// TIA Portal V19 export
FUNCTION_BLOCK "Main Control"   // FB1, LAD
{ S7_Optimized_Access := 'TRUE' }
// stored: MemoryReserve 100, SetENOAutomatically false
   VAR
      store : Bool;
   END_VAR
   VAR_TEMP   // added for the SCL form of the ladder/FBD networks
      _w1 : Bool;
      _w2 : Bool;
   END_VAR
BEGIN

REGION Network 1: Control Auto Run
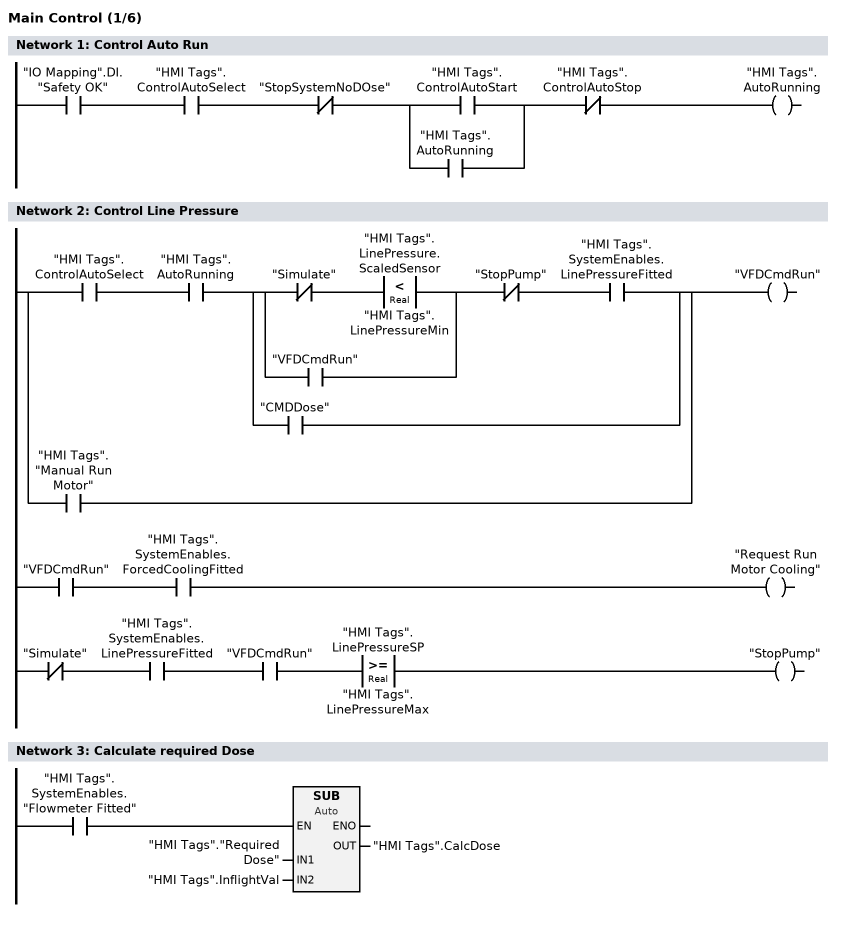
   RUNG wire#powerrail
      Contact( "IO Mapping".DI."Safety OK" )
      Contact( "HMI Tags".ControlAutoSelect )
      I_Contact( "StopSystemNoDOse" )
      wire#w1
      Contact( "HMI Tags".ControlAutoStart )
      wire#w2
      I_Contact( "HMI Tags".ControlAutoStop )
      Coil( "HMI Tags".AutoRunning )
   END_RUNG
   RUNG wire#w1
      Contact( "HMI Tags".AutoRunning )
   END_RUNG wire#w2
   // the same network as SCL:
   "HMI Tags".AutoRunning := "IO Mapping".DI."Safety OK" AND "HMI Tags".ControlAutoSelect AND NOT "StopSystemNoDOse" AND ("HMI Tags".ControlAutoStart OR "HMI Tags".AutoRunning) AND NOT "HMI Tags".ControlAutoStop;
END_REGION

REGION Network 2: Control Line Pressure
   RUNG wire#powerrail
      Contact( "HMI Tags".ControlAutoSelect )
      Contact( "HMI Tags".AutoRunning )
      wire#w1
      I_Contact( "Simulate" )
      { S7_Templates := "SrcType := Real" } LT_Contact(in1 := "HMI Tags".LinePressure.ScaledSensor, in2 := "HMI Tags".LinePressureMin)
      wire#w2
      I_Contact( "StopPump" )
      Contact( "HMI Tags".SystemEnables.LinePressureFitted )
      wire#w3
      Coil( "VFDCmdRun" )
   END_RUNG
   RUNG wire#w1
      Contact( "VFDCmdRun" )
   END_RUNG wire#w2
   RUNG wire#w1
      Contact( "CMDDose" )
   END_RUNG wire#w3
   RUNG wire#powerrail
      Contact( "HMI Tags"."Manual Run Motor" )
   END_RUNG wire#w3
   RUNG wire#powerrail
      Contact( "VFDCmdRun" )
      Contact( "HMI Tags".SystemEnables.ForcedCoolingFitted )
      Coil( "Request Run Motor Cooling" )
   END_RUNG
   RUNG wire#powerrail
      I_Contact( "Simulate" )
      Contact( "HMI Tags".SystemEnables.LinePressureFitted )
      Contact( "VFDCmdRun" )
      { S7_Templates := "SrcType := Real" } GE_Contact(in1 := "HMI Tags".LinePressureSP, in2 := "HMI Tags".LinePressureMax)
      Coil( "StopPump" )
   END_RUNG
   // the same network as SCL:
   "VFDCmdRun" := ("HMI Tags".ControlAutoSelect AND "HMI Tags".AutoRunning AND ((((NOT "Simulate" AND ("HMI Tags".LinePressure.ScaledSensor < "HMI Tags".LinePressureMin)) OR "VFDCmdRun") AND NOT "StopPump" AND "HMI Tags".SystemEnables.LinePressureFitted) OR "CMDDose")) OR "HMI Tags"."Manual Run Motor";
   "Request Run Motor Cooling" := "VFDCmdRun" AND "HMI Tags".SystemEnables.ForcedCoolingFitted;
   "StopPump" := NOT "Simulate" AND "HMI Tags".SystemEnables.LinePressureFitted AND "VFDCmdRun" AND ("HMI Tags".LinePressureSP >= "HMI Tags".LinePressureMax);
END_REGION

REGION Network 3: Calculate required Dose
   RUNG wire#powerrail
      Contact( "HMI Tags".SystemEnables."Flowmeter Fitted" )
      Sub(in1 := "HMI Tags"."Required Dose", in2 := "HMI Tags".InflightVal, out => "HMI Tags".CalcDose)
   END_RUNG
   // the same network as SCL:
   IF "HMI Tags".SystemEnables."Flowmeter Fitted" THEN
       "HMI Tags".CalcDose := "HMI Tags"."Required Dose" - "HMI Tags".InflightVal;
   END_IF;
END_REGION

REGION Network 4: Open Valves to Dose
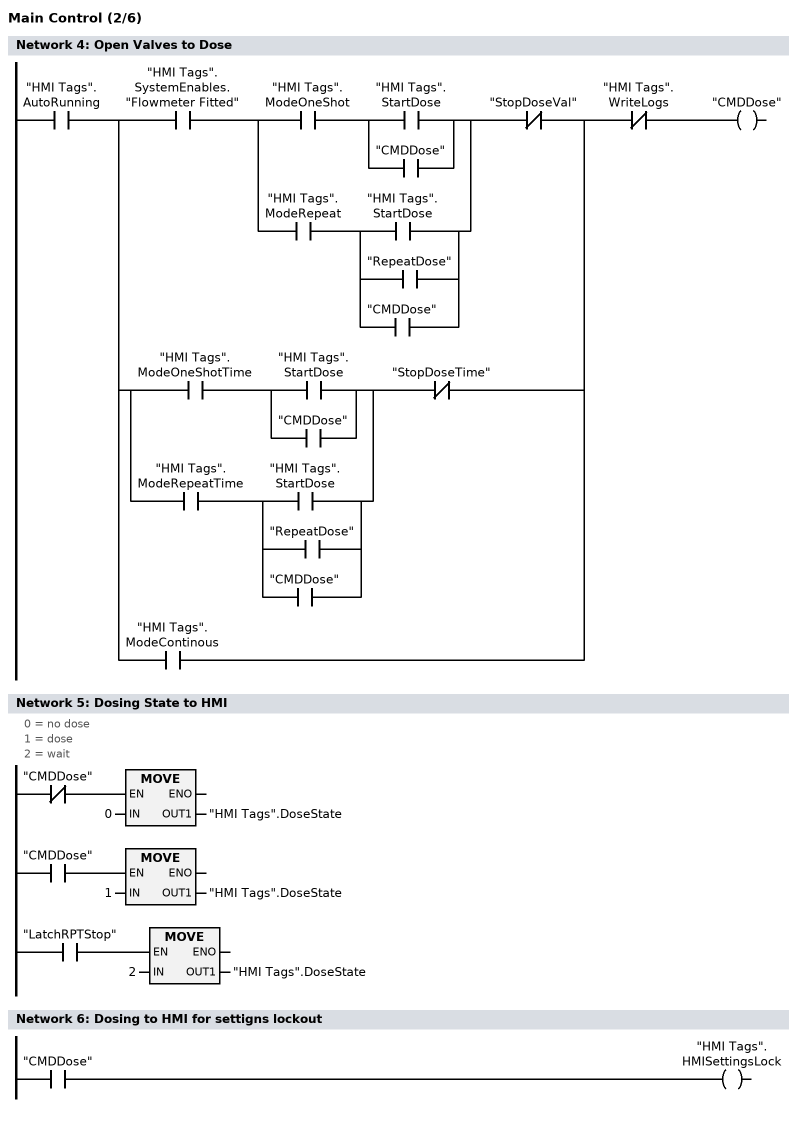
   RUNG wire#powerrail
      Contact( "HMI Tags".AutoRunning )
      wire#w1
      Contact( "HMI Tags".SystemEnables."Flowmeter Fitted" )
      wire#w2
      Contact( "HMI Tags".ModeOneShot )
      wire#w3
      Contact( "HMI Tags".StartDose )
      wire#w4
      I_Contact( "StopDoseVal" )
      wire#w6
      I_Contact( "HMI Tags".WriteLogs )
      Coil( "CMDDose" )
   END_RUNG
   RUNG wire#w3
      Contact( "CMDDose" )
   END_RUNG wire#w4
   RUNG wire#w2
      Contact( "HMI Tags".ModeRepeat )
      wire#w5
      Contact( "HMI Tags".StartDose )
   END_RUNG wire#w4
   RUNG wire#w5
      Contact( "RepeatDose" )
   END_RUNG wire#w4
   RUNG wire#w5
      Contact( "CMDDose" )
   END_RUNG wire#w4
   RUNG wire#w1
      Contact( "HMI Tags".ModeOneShotTime )
      wire#w7
      Contact( "HMI Tags".StartDose )
      wire#w8
      I_Contact( "StopDoseTime" )
   END_RUNG wire#w6
   RUNG wire#w7
      Contact( "CMDDose" )
   END_RUNG wire#w8
   RUNG wire#w1
      Contact( "HMI Tags".ModeRepeatTime )
      wire#w9
      Contact( "HMI Tags".StartDose )
   END_RUNG wire#w8
   RUNG wire#w9
      Contact( "RepeatDose" )
   END_RUNG wire#w8
   RUNG wire#w9
      Contact( "CMDDose" )
   END_RUNG wire#w8
   RUNG wire#w1
      Contact( "HMI Tags".ModeContinous )
   END_RUNG wire#w6
   // the same network as SCL:
   "CMDDose" := "HMI Tags".AutoRunning AND (("HMI Tags".SystemEnables."Flowmeter Fitted" AND (("HMI Tags".ModeOneShot AND ("HMI Tags".StartDose OR "CMDDose")) OR ("HMI Tags".ModeRepeat AND ("HMI Tags".StartDose OR "RepeatDose" OR "CMDDose"))) AND NOT "StopDoseVal") OR ((("HMI Tags".ModeOneShotTime AND ("HMI Tags".StartDose OR "CMDDose")) OR ("HMI Tags".ModeRepeatTime AND ("HMI Tags".StartDose OR "RepeatDose" OR "CMDDose"))) AND NOT "StopDoseTime") OR "HMI Tags".ModeContinous) AND NOT "HMI Tags".WriteLogs;
END_REGION

REGION Network 5: Dosing State to HMI
   // 0 = no dose
   // 1 = dose
   // 2 = wait
   RUNG wire#powerrail
      I_Contact( "CMDDose" )
      Move(in := 0, out1 => "HMI Tags".DoseState)
   END_RUNG
   RUNG wire#powerrail
      Contact( "CMDDose" )
      Move(in := 1, out1 => "HMI Tags".DoseState)
   END_RUNG
   RUNG wire#powerrail
      Contact( "LatchRPTStop" )
      Move(in := 2, out1 => "HMI Tags".DoseState)
   END_RUNG
   // the same network as SCL:
   IF NOT "CMDDose" THEN "HMI Tags".DoseState := 0; END_IF;
   IF "CMDDose" THEN "HMI Tags".DoseState := 1; END_IF;
   IF "LatchRPTStop" THEN "HMI Tags".DoseState := 2; END_IF;
END_REGION

REGION Network 6: Dosing to HMI for settigns lockout
   RUNG wire#powerrail
      Contact( "CMDDose" )
      Coil( "HMI Tags".HMISettingsLock )
   END_RUNG
   // the same network as SCL:
   "HMI Tags".HMISettingsLock := "CMDDose";
END_REGION

REGION Network 7: Command the flowmeter to count
   // This should start the flowmeter counting slightly ahead of opening the valves.
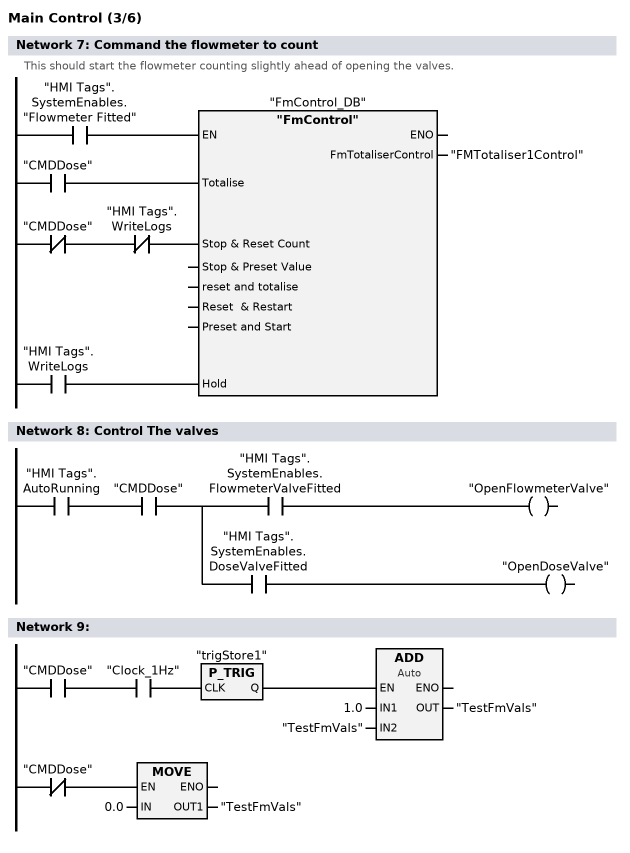
   RUNG wire#powerrail
      Contact( "HMI Tags".SystemEnables."Flowmeter Fitted" )
      "FmControl_DB"(Totalise := wire#w1, "Stop & Reset Count" := wire#w2, Hold := wire#w3, "Stop & Preset Value" :=, "reset and totalise" :=, "Reset  & Restart" :=, "Preset and Start" :=, FmTotaliserControl => "FMTotaliser1Control")
   END_RUNG
   RUNG wire#powerrail
      Contact( "CMDDose" )
   END_RUNG wire#w1
   RUNG wire#powerrail
      I_Contact( "CMDDose" )
      I_Contact( "HMI Tags".WriteLogs )
   END_RUNG wire#w2
   RUNG wire#powerrail
      Contact( "HMI Tags".WriteLogs )
   END_RUNG wire#w3
   // the same network as SCL:
   IF "HMI Tags".SystemEnables."Flowmeter Fitted" THEN
       "FmControl_DB"(Totalise := "CMDDose",   // "FmControl"
                      "Stop & Reset Count" := NOT "CMDDose" AND NOT "HMI Tags".WriteLogs,
                      Hold := "HMI Tags".WriteLogs,
                      FmTotaliserControl => "FMTotaliser1Control");
   END_IF;
END_REGION

REGION Network 8: Control The valves
   RUNG wire#powerrail
      Contact( "HMI Tags".AutoRunning )
      Contact( "CMDDose" )
      wire#w1
      Contact( "HMI Tags".SystemEnables.FlowmeterValveFitted )
      Coil( "OpenFlowmeterValve" )
   END_RUNG
   RUNG wire#w1
      Contact( "HMI Tags".SystemEnables.DoseValveFitted )
      Coil( "OpenDoseValve" )
   END_RUNG
   // the same network as SCL:
   #_w1 := "HMI Tags".AutoRunning AND "CMDDose";
   "OpenFlowmeterValve" := #_w1 AND "HMI Tags".SystemEnables.FlowmeterValveFitted;
   "OpenDoseValve" := #_w1 AND "HMI Tags".SystemEnables.DoseValveFitted;
END_REGION

REGION Network 9
   RUNG wire#powerrail
      Contact( "CMDDose" )
      Contact( "Clock_1Hz" )
      P_Trig( "trigStore1" )
      Add(in1 := 1.0, in2 := "TestFmVals", out => "TestFmVals")
   END_RUNG
   RUNG wire#powerrail
      I_Contact( "CMDDose" )
      Move(in := 0.0, out1 => "TestFmVals")
   END_RUNG
   // the same network as SCL:
   #_w1 := "CMDDose" AND "Clock_1Hz";
   #_w2 := #_w1 AND NOT "trigStore1";   // rising edge
   "trigStore1" := #_w1;
   IF #_w2 THEN "TestFmVals" := 1.0 + "TestFmVals"; END_IF;
   IF NOT "CMDDose" THEN "TestFmVals" := 0.0; END_IF;
END_REGION

REGION Network 10: Wait for flow Value OneShot value or time
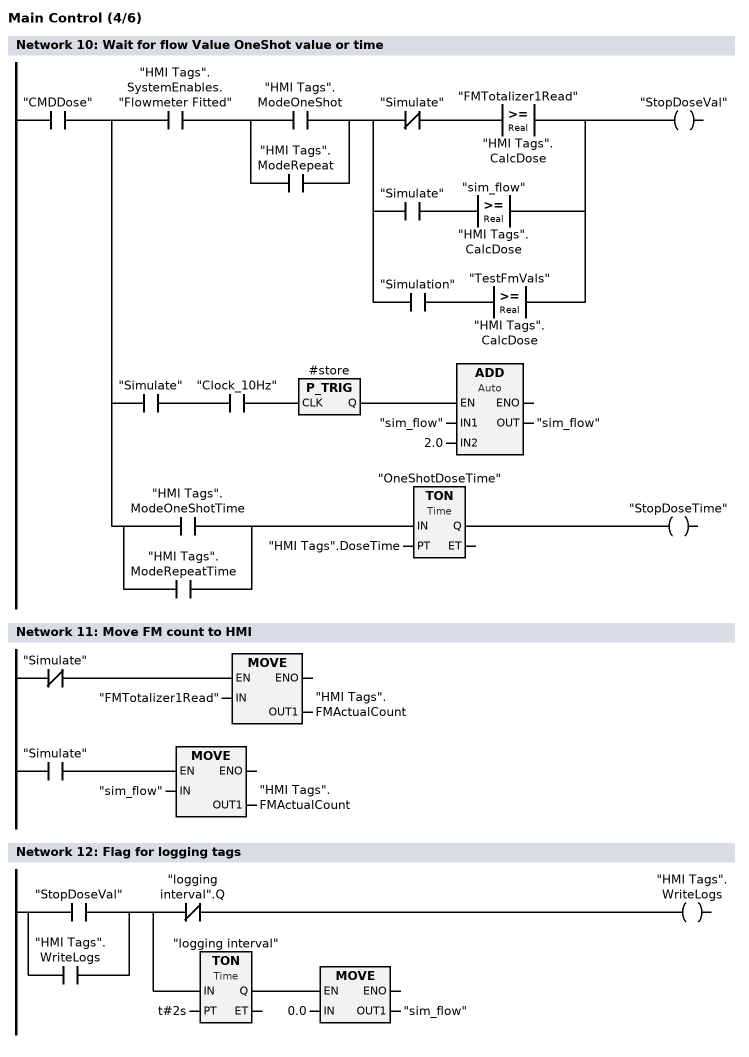
   RUNG wire#powerrail
      Contact( "CMDDose" )
      wire#w1
      Contact( "HMI Tags".SystemEnables."Flowmeter Fitted" )
      wire#w2
      Contact( "HMI Tags".ModeOneShot )
      wire#w3
      I_Contact( "Simulate" )
      { S7_Templates := "SrcType := Real" } GE_Contact(in1 := "FMTotalizer1Read", in2 := "HMI Tags".CalcDose)
      wire#w4
      Coil( "StopDoseVal" )
   END_RUNG
   RUNG wire#w2
      Contact( "HMI Tags".ModeRepeat )
   END_RUNG wire#w3
   RUNG wire#w3
      Contact( "Simulate" )
      { S7_Templates := "SrcType := Real" } GE_Contact(in1 := "sim_flow", in2 := "HMI Tags".CalcDose)
   END_RUNG wire#w4
   RUNG wire#w3
      Contact( "Simulation" )
      { S7_Templates := "SrcType := Real" } GE_Contact(in1 := "TestFmVals", in2 := "HMI Tags".CalcDose)
   END_RUNG wire#w4
   RUNG wire#w1
      Contact( "Simulate" )
      Contact( "Clock_10Hz" )
      P_Trig( #store )
      Add(in1 := "sim_flow", in2 := 2.0, out => "sim_flow")
   END_RUNG
   RUNG wire#w1
      Contact( "HMI Tags".ModeOneShotTime )
      wire#w5
      { S7_Templates := "time_type := Time" } "OneShotDoseTime".TON(pt := "HMI Tags".DoseTime, et =>)
      Coil( "StopDoseTime" )
   END_RUNG
   RUNG wire#w1
      Contact( "HMI Tags".ModeRepeatTime )
   END_RUNG wire#w5
   // the same network as SCL:
   "StopDoseVal" := "CMDDose" AND "HMI Tags".SystemEnables."Flowmeter Fitted" AND ("HMI Tags".ModeOneShot OR "HMI Tags".ModeRepeat) AND ((NOT "Simulate" AND ("FMTotalizer1Read" >= "HMI Tags".CalcDose)) OR ("Simulate" AND ("sim_flow" >= "HMI Tags".CalcDose)) OR ("Simulation" AND ("TestFmVals" >= "HMI Tags".CalcDose)));
   #_w1 := "CMDDose" AND "Simulate" AND "Clock_10Hz";
   #_w2 := #_w1 AND NOT #store;   // rising edge
   #store := #_w1;
   IF #_w2 THEN "sim_flow" := "sim_flow" + 2.0; END_IF;
   "OneShotDoseTime".TON(IN := "CMDDose" AND ("HMI Tags".ModeOneShotTime OR "HMI Tags".ModeRepeatTime),
                         PT := "HMI Tags".DoseTime);
   "StopDoseTime" := "OneShotDoseTime".Q;
END_REGION

REGION Network 11: Move FM count to HMI
   RUNG wire#powerrail
      I_Contact( "Simulate" )
      Move(in := "FMTotalizer1Read", out1 => "HMI Tags".FMActualCount)
   END_RUNG
   RUNG wire#powerrail
      Contact( "Simulate" )
      Move(in := "sim_flow", out1 => "HMI Tags".FMActualCount)
   END_RUNG
   // the same network as SCL:
   IF NOT "Simulate" THEN "HMI Tags".FMActualCount := "FMTotalizer1Read"; END_IF;
   IF "Simulate" THEN "HMI Tags".FMActualCount := "sim_flow"; END_IF;
END_REGION

REGION Network 12: Flag for logging tags
   RUNG wire#powerrail
      Contact( "StopDoseVal" )
      wire#w1
      I_Contact( "logging interval".Q )
      Coil( "HMI Tags".WriteLogs )
   END_RUNG
   RUNG wire#powerrail
      Contact( "HMI Tags".WriteLogs )
   END_RUNG wire#w1
   RUNG wire#w1
      { S7_Templates := "time_type := Time" } "logging interval".TON(pt := t#2s, et =>)
      Move(in := 0.0, out1 => "sim_flow")
   END_RUNG
   // the same network as SCL:
   #_w1 := "StopDoseVal" OR "HMI Tags".WriteLogs;
   "HMI Tags".WriteLogs := #_w1 AND NOT "logging interval".Q;
   "logging interval".TON(IN := #_w1, PT := t#2s);
   IF "logging interval".Q THEN "sim_flow" := 0.0; END_IF;
END_REGION

REGION Network 13: Repeat Dose After Time
   // Latch dose start and dose stop for repeat doses then unlatch on the next dose
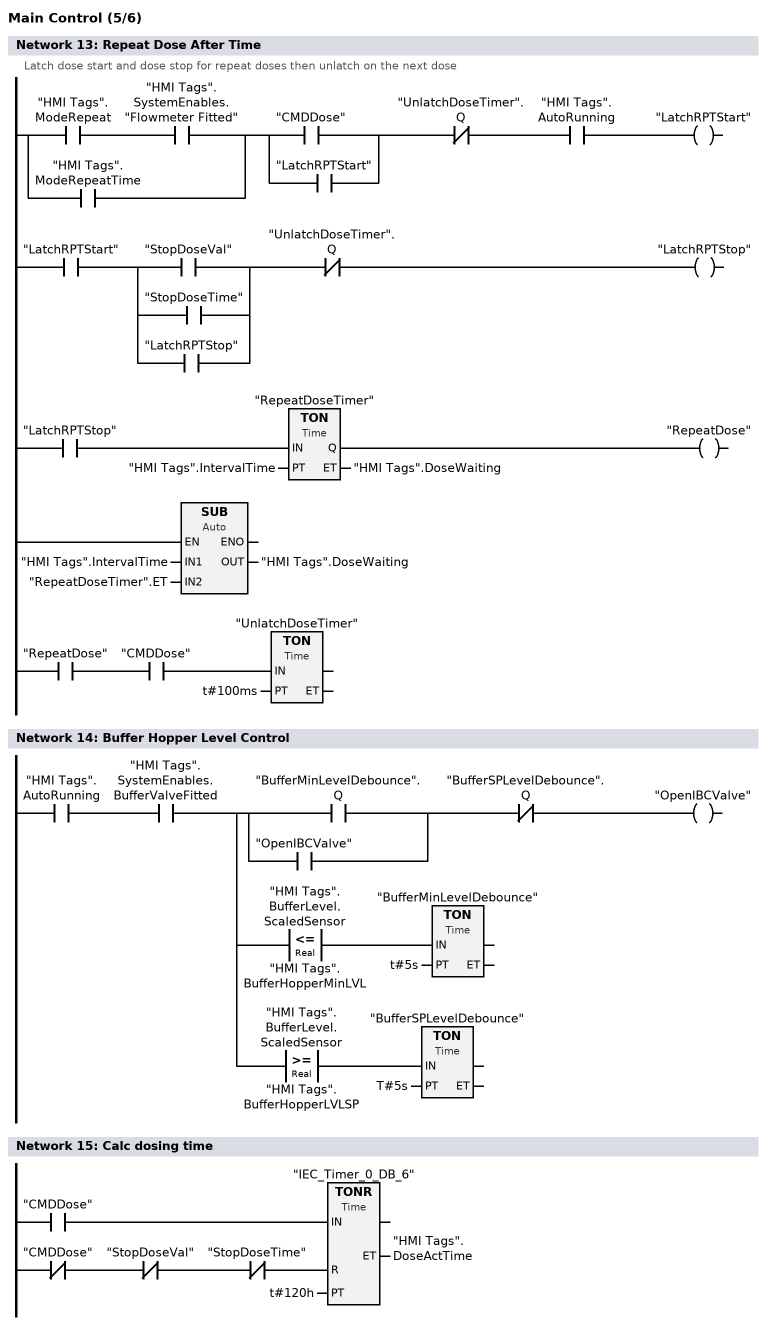
   RUNG wire#powerrail
      Contact( "HMI Tags".ModeRepeat )
      Contact( "HMI Tags".SystemEnables."Flowmeter Fitted" )
      wire#w1
      Contact( "CMDDose" )
      wire#w2
      I_Contact( "UnlatchDoseTimer".Q )
      Contact( "HMI Tags".AutoRunning )
      Coil( "LatchRPTStart" )
   END_RUNG
   RUNG wire#powerrail
      Contact( "HMI Tags".ModeRepeatTime )
   END_RUNG wire#w1
   RUNG wire#w1
      Contact( "LatchRPTStart" )
   END_RUNG wire#w2
   RUNG wire#powerrail
      Contact( "LatchRPTStart" )
      wire#w3
      Contact( "StopDoseVal" )
      wire#w4
      I_Contact( "UnlatchDoseTimer".Q )
      Coil( "LatchRPTStop" )
   END_RUNG
   RUNG wire#w3
      Contact( "StopDoseTime" )
   END_RUNG wire#w4
   RUNG wire#w3
      Contact( "LatchRPTStop" )
   END_RUNG wire#w4
   RUNG wire#powerrail
      Contact( "LatchRPTStop" )
      { S7_Templates := "time_type := Time" } "RepeatDoseTimer".TON(pt := "HMI Tags".IntervalTime, et => "HMI Tags".DoseWaiting)
      Coil( "RepeatDose" )
   END_RUNG
   RUNG wire#powerrail
      Sub(in1 := "HMI Tags".IntervalTime, in2 := "RepeatDoseTimer".ET, out => "HMI Tags".DoseWaiting)
   END_RUNG
   RUNG wire#powerrail
      Contact( "RepeatDose" )
      Contact( "CMDDose" )
      { S7_Templates := "time_type := Time" } "UnlatchDoseTimer".TON(pt := t#100ms, et =>)
   END_RUNG
   // the same network as SCL:
   "LatchRPTStart" := (("HMI Tags".ModeRepeat AND "HMI Tags".SystemEnables."Flowmeter Fitted") OR "HMI Tags".ModeRepeatTime) AND ("CMDDose" OR "LatchRPTStart") AND NOT "UnlatchDoseTimer".Q AND "HMI Tags".AutoRunning;
   "LatchRPTStop" := "LatchRPTStart" AND ("StopDoseVal" OR "StopDoseTime" OR "LatchRPTStop") AND NOT "UnlatchDoseTimer".Q;
   "RepeatDoseTimer".TON(IN := "LatchRPTStop", PT := "HMI Tags".IntervalTime, ET => "HMI Tags".DoseWaiting);
   "RepeatDose" := "RepeatDoseTimer".Q;
   "HMI Tags".DoseWaiting := "HMI Tags".IntervalTime - "RepeatDoseTimer".ET;
   "UnlatchDoseTimer".TON(IN := "RepeatDose" AND "CMDDose", PT := t#100ms);
END_REGION

REGION Network 14: Buffer Hopper Level Control
   RUNG wire#powerrail
      Contact( "HMI Tags".AutoRunning )
      Contact( "HMI Tags".SystemEnables.BufferValveFitted )
      wire#w1
      Contact( "BufferMinLevelDebounce".Q )
      wire#w2
      I_Contact( "BufferSPLevelDebounce".Q )
      Coil( "OpenIBCValve" )
   END_RUNG
   RUNG wire#w1
      Contact( "OpenIBCValve" )
   END_RUNG wire#w2
   RUNG wire#w1
      { S7_Templates := "SrcType := Real" } LE_Contact(in1 := "HMI Tags".BufferLevel.ScaledSensor, in2 := "HMI Tags".BufferHopperMinLVL)
      { S7_Templates := "time_type := Time" } "BufferMinLevelDebounce".TON(pt := t#5s, et =>)
   END_RUNG
   RUNG wire#w1
      { S7_Templates := "SrcType := Real" } GE_Contact(in1 := "HMI Tags".BufferLevel.ScaledSensor, in2 := "HMI Tags".BufferHopperLVLSP)
      { S7_Templates := "time_type := Time" } "BufferSPLevelDebounce".TON(pt := T#5s, et =>)
   END_RUNG
   // the same network as SCL:
   #_w1 := "HMI Tags".AutoRunning AND "HMI Tags".SystemEnables.BufferValveFitted;
   "OpenIBCValve" := #_w1 AND ("BufferMinLevelDebounce".Q OR "OpenIBCValve") AND NOT "BufferSPLevelDebounce".Q;
   "BufferMinLevelDebounce".TON(IN := #_w1 AND ("HMI Tags".BufferLevel.ScaledSensor <= "HMI Tags".BufferHopperMinLVL),
                           PT := t#5s);
   "BufferSPLevelDebounce".TON(IN := #_w1 AND ("HMI Tags".BufferLevel.ScaledSensor >= "HMI Tags".BufferHopperLVLSP),
                           PT := T#5s);
END_REGION

REGION Network 15: Calc dosing time
   RUNG wire#powerrail
      Contact( "CMDDose" )
      { S7_Templates := "time_type := Time" } "IEC_Timer_0_DB_6".TONR(r := wire#w1, pt := t#120h, et => "HMI Tags".DoseActTime)
   END_RUNG
   RUNG wire#powerrail
      I_Contact( "CMDDose" )
      I_Contact( "StopDoseVal" )
      I_Contact( "StopDoseTime" )
   END_RUNG wire#w1
   // the same network as SCL:
   "IEC_Timer_0_DB_6".TONR(IN := "CMDDose",
                           R := NOT "CMDDose" AND NOT "StopDoseVal" AND NOT "StopDoseTime",
                           PT := t#120h,
                           ET => "HMI Tags".DoseActTime);
END_REGION

REGION Network 16: flowmeter Temperature
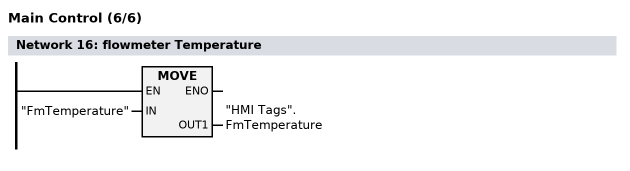
   RUNG wire#powerrail
      Move(in := "FmTemperature", out1 => "HMI Tags".FmTemperature)
   END_RUNG
   // the same network as SCL:
   "HMI Tags".FmTemperature := "FmTemperature";
END_REGION
END_FUNCTION_BLOCK
